(* IEC 61131-3 sources: CodesysTest/alpha/export/FBs/Components/Load Plate/FB_BaseLoadPlate.pou, 6 files *)

(* ---- FB_BaseLoadPlate.pou.st ---- *)
(*#-#-#-#-#-#-#-#-#-#---Declaration---#-#-#-#-#-#-#-#-#-#-#-#-#*)

FUNCTION_BLOCK FB_BaseLoadPlate EXTENDS FB_BaseComponent
VAR_INPUT
	inUse : BOOL;
	faultActive : BOOL;
	dischargeOnFault : BOOL;
	inLoadingPosition : BOOL;
	inDischargePosition : BOOL;
	switchedPowerON : BOOL;
	faultsEnabled : BOOL;
	triggerDwell : REAL;
	triggerDelay : REAL;
    shakerEnable : BOOL;
	shakerDwell : REAL;
	shakerDelay : REAL;
	shakerOnDwell : REAL;
	shakerOffDwell : REAL;
	shakeStart : SHAKER_START_SELECTION;
	disabledPosition : PackageEjectionDisabledPosition;
END_VAR
VAR_OUTPUT
	moveToDischargePosition : BOOL;
	moveToLoadingPositon : BOOL;
	failedToExtend : BOOL;
	failedToRetract : BOOL;
END_VAR
VAR
	_faultActiveONS : FB_ONS;
	_faultTime : TIME := T#2500MS;
	_shake : BOOL;
	_shaking : BOOL;
	_trigger : BOOL;
	_manualOn : BOOL;
	_manualOff : BOOL;
	_shaker : Util.BLINK;
	_shakerDelayTimer : Standard.TON;
	_shakerDwellTimer : Standard.TON;
	_triggerDelayTimer : Standard.TON;
	_triggerDwellTimer : Standard.TON;
	_extendFaultTimer : Standard.TON;
	_retractFaultTimer : Standard.TON;
	_triggerONS : FB_ONS;
	_shakeONS : FB_ONS;
	_state : LOAD_PLATE_STATE;
	_inUseONS : FB_ONS;
	_switchedPowerOnONS : FB_ONS;
	_disabledPositionHasUpdated : BOOL;
	_previousDisabledPosition : PackageEjectionDisabledPosition;
	_updateNotInUsePosition : BOOL;
END_VAR
(*#-#-#-#-#-#-#-#-#-#---Implementation---#-#-#-#-#-#-#-#-#-#-#-#-#*)

//
//  FB_BaseLoadPlate
//  FBs/Components/LoadPlate/FB_BaseLoadPlate
//
//  Created by Evan Ische on 6/19/2021.
//  Copyright (C) 2021 Sharp Packaging Systems By Pregis. All rights reserved.
//

SUPER^();

// Null Parameters on reset of cycle completion
IF _triggerDwellTimer.Q OR resetONS.Q THEN
	_trigger := FALSE;
	_shaking := FALSE;
	_shake := FALSE;
	_shakerDelayTimer.IN := FALSE;
	_shakerDwellTimer.IN := FALSE;
	_extendFaultTimer.IN := FALSE;
	_retractFaultTimer.IN := FALSE;
	_state := LOAD_PLATE_STATE.Idle;
END_IF

//
_inUseONS(CLK := inUse);

//
_shakeONS(CLK := _shaker.OUT);

//
_triggerONS(CLK := _triggerDelayTimer.Q);

//
_faultActiveONS(CLK := faultActive);

//
_disabledPositionHasUpdated := FALSE;
IF disabledPosition <> _previousDisabledPosition THEN
	_disabledPositionHasUpdated := TRUE;
	_previousDisabledPosition := disabledPosition;
END_IF
_switchedPowerOnONS(CLK := switchedPowerON);

//
_updateNotInUsePosition := (_switchedPowerOnONS.OSR OR _disabledPositionHasUpdated OR _inUseONS.OSF);
IF _manualOn
	OR ((_triggerONS.OSR OR _shakeONS.OSF OR (_faultActiveONS.OSR AND switchedPowerON AND dischargeOnFault)) AND inUse)
	OR (_updateNotInUsePosition AND DischargePositionWhileDisabled AND NOT inUse)
	THEN
		moveToDischargePosition := TRUE;
		_manualOn := FALSE;
ELSIF _manualOff
	OR (((_triggerONS.OSF AND NOT faultActive) OR _shakeONS.OSR OR _inUseONS.OSR OR resetONS.Q) AND inUse)
	OR (_updateNotInUsePosition AND LoadingPositionWhileDisabled AND NOT inUse)
	THEN
		moveToDischargePosition := FALSE;
		_manualOff := FALSE;
END_IF
moveToLoadingPositon := NOT moveToDischargePosition;

// Counts the time between telling an actuator to move positions, and when it gets to the new position. If Timer finished, fault.
_extendFaultTimer(
	IN := moveToLoadingPositon AND NOT inLoadingPosition AND faultsEnabled AND NOT resetONS.Q,
	PT := _faultTime,
	 Q => failedToExtend);

_retractFaultTimer(
	IN := moveToDischargePosition AND NOT inDischargePosition AND faultsEnabled AND NOT resetONS.Q,
	PT := _faultTime,
	 Q => failedToRetract);

// How Long To Wait Before Going Active
_triggerDelayTimer(
	IN := _trigger,
	PT := TO_TIME(triggerDelay * 1000));

// Retract Duration
_triggerDwellTimer(
	IN := _triggerDelayTimer.Q,
	PT := TO_TIME(triggerDwell * 1000));

//
_shaker(
	TIMEHIGH := TO_TIME(shakerOnDwell * 1000),
	TIMELOW := TO_TIME(shakerOffDwell * 1000));
_shakerDelayTimer(PT := TO_TIME(shakerDelay * 1000));
_shakerDwellTimer(PT := TO_TIME(shakerDwell * 1000));

//
CASE _state OF
	LOAD_PLATE_STATE.Idle:
		IF _shake THEN
			_shake := FALSE;
			_state := LOAD_PLATE_STATE.Shake;
		END_IF

	LOAD_PLATE_STATE.Shake:
		_shakerDelayTimer.IN := TRUE;
		IF _shakerDelayTimer.Q THEN
			_shakerDelayTimer.IN := FALSE;
			_state := LOAD_PLATE_STATE.Shaking;
		END_IF

	LOAD_PLATE_STATE.Shaking:
		// Starts Shaker
		_shaker.ENABLE := TRUE;
		_shakerDwellTimer.IN := TRUE;
		IF _shakerDwellTimer.Q THEN
			// Ends Shaker
			_shaker.ENABLE := FALSE;
			_shakerDwellTimer.IN := FALSE;
			_state := LOAD_PLATE_STATE.Shaked;
		END_IF

	LOAD_PLATE_STATE.Shaked:
		IF inLoadingPosition THEN
			_state := LOAD_PLATE_STATE.Idle;
		ELSE
			IF NOT inLoadingPosition THEN
				_manualOff := TRUE;
			END_IF
		END_IF
END_CASE

(* ---- ManualOff.m.st ---- *)
(*#-#-#-#-#-#-#-#-#-#---Declaration---#-#-#-#-#-#-#-#-#-#-#-#-#*)

METHOD ManualOff
VAR_INPUT
END_VAR
(*#-#-#-#-#-#-#-#-#-#---Implementation---#-#-#-#-#-#-#-#-#-#-#-#-#*)

IF enable THEN
	_manualOff := TRUE;
END_IF

(* ---- ManualON.m.st ---- *)
(*#-#-#-#-#-#-#-#-#-#---Declaration---#-#-#-#-#-#-#-#-#-#-#-#-#*)

METHOD ManualON
VAR_INPUT
END_VAR
(*#-#-#-#-#-#-#-#-#-#---Implementation---#-#-#-#-#-#-#-#-#-#-#-#-#*)

IF enable THEN
	_manualOn := TRUE;
END_IF

(* ---- moveToDischargePos.m.st ---- *)
(*#-#-#-#-#-#-#-#-#-#---Declaration---#-#-#-#-#-#-#-#-#-#-#-#-#*)

METHOD moveToDischargePos
VAR_INPUT
END_VAR
(*#-#-#-#-#-#-#-#-#-#---Implementation---#-#-#-#-#-#-#-#-#-#-#-#-#*)

IF enable THEN
	_manualOn := TRUE;
END_IF

(* ---- moveToLoadingPos.m.st ---- *)
(*#-#-#-#-#-#-#-#-#-#---Declaration---#-#-#-#-#-#-#-#-#-#-#-#-#*)

METHOD moveToLoadingPos
VAR_INPUT
END_VAR
(*#-#-#-#-#-#-#-#-#-#---Implementation---#-#-#-#-#-#-#-#-#-#-#-#-#*)

IF enable THEN
	_manualOff := TRUE;
END_IF

(* ---- Shake.m.st ---- *)
(*#-#-#-#-#-#-#-#-#-#---Declaration---#-#-#-#-#-#-#-#-#-#-#-#-#*)

METHOD Shake
VAR_INPUT
END_VAR
(*#-#-#-#-#-#-#-#-#-#---Implementation---#-#-#-#-#-#-#-#-#-#-#-#-#*)

IF enable AND shakerEnable AND (shakerDwell > 0) AND inUse THEN
	_shake := TRUE;
END_IF
